RESOURCE_TYPE _Core102
  (* Standard: 61499-2 *)
  (* Version 0.1, 2017-00-01, hpea485, UOA *)
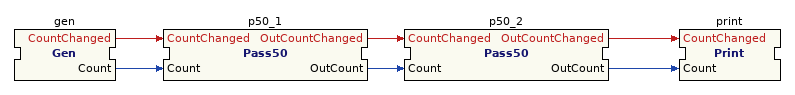
  FBS
    gen : Gen;
    print : Print;
    p50_1 : Pass50;
    p50_2 : Pass50;
  END_FBS
  EVENT_CONNECTIONS
    gen.CountChanged TO p50_1.CountChanged;
    p50_1.OutCountChanged TO p50_2.CountChanged;
    p50_2.OutCountChanged TO print.CountChanged;
  END_CONNECTIONS
  DATA_CONNECTIONS
    gen.Count TO p50_1.Count;
    p50_1.OutCount TO p50_2.Count;
    p50_2.OutCount TO print.Count;
  END_CONNECTIONS
END_RESOURCE_TYPE
